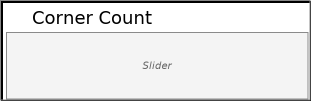
VISUALIZATION InputNumSlider  // 311x101
    Rectangle (1,1 310x100)
    Slider (6,32 302x67), variable: MAIN.FB_FigureGenerator.nCornerCountInp, scale 3..13
    Label (17,3 150x30), "Corner Count"
END_VISUALIZATION

(* stored: Version 1.1.0.1, ProductVersion 3.1.4024.12
   Visu InputNumSlider: Id {96a97254-8599-42e3-bfab-09ee7a10b194} *)
